(* PLC project Untitled1, Beckhoff Automation GmbH TF6420 Database Server Query Analyser 1.0.0.0 *)
(* stored: creationDateTime 2016-04-21T15:04:54, modificationDateTime 2016-04-21T15:04:54 *)

TYPE ST_DB_EV : STRUCT
  id : DINT;
  Timestamp : DT;
  Name : STRING(45);
  IstDruck : REAL;
  IstTemp : REAL;
  SaugTemp : REAL;
  VerdampfTemp : REAL;
  VerdampfDruck : REAL;
  UberhitzungTemp : REAL;
  VentilOffnung : REAL;
  RegelSollwert : REAL;
  Ventilposition : REAL;
  AktKuhlleistung : REAL;
END_STRUCT;
END_TYPE
